{attribute 'GeneratedUsingTerminal: KL8528'}
{attribute addProperty BoxType "KL8528"}
{attribute addProperty Id "Channel_1AT %Q*Channel_D490E9730"}
{attribute addProperty CRC "1940487873"}
{attribute addProperty Size "0"}
TYPE KL8528_73A97EC1 :
STRUCT
	{attribute addProperty Name "Channel_1"}
	Channel_1 : Channel_D490E973;
END_STRUCT
END_TYPE

(* stored: Version 1.2.0.0, ProductVersion 3.1.4024.9
   DUT KL8528_73A97EC1: Id {f9224094-a404-41b1-af9b-30e1dccaed7a} *)
